// TIA Portal V16 export
// export: Created 2021-08-26T13:23:50.3138984Z, ExportSetting WithDefaults, DisplayName Totally Integrated Automation Portal, DisplayVersion V16 Update 4, DisplayName TIA Portal Version Control Interface, DisplayVersion V16 Update 2, DisplayName TIA Portal Openness, DisplayVersion V16 Update 4, DisplayName STEP 7 Professional, DisplayVersion V16 Update 4, DisplayName STEP 7 Safety, DisplayVersion V16, DisplayName WinCC Advanced, DisplayVersion V16 Update 4
FUNCTION "funkcja1" : Void   // FC1, LAD
TITLE = taki oto jest tytul bloku
{ S7_Optimized_Access := 'TRUE' }
VERSION : 0.1
// komentarz bloku
// stored: AutoNumber false, IsIECCheckEnabled false, SetENOAutomatically false, UDAEnableTagReadback false
BEGIN

REGION Network 1: bardzo ważny komentarz
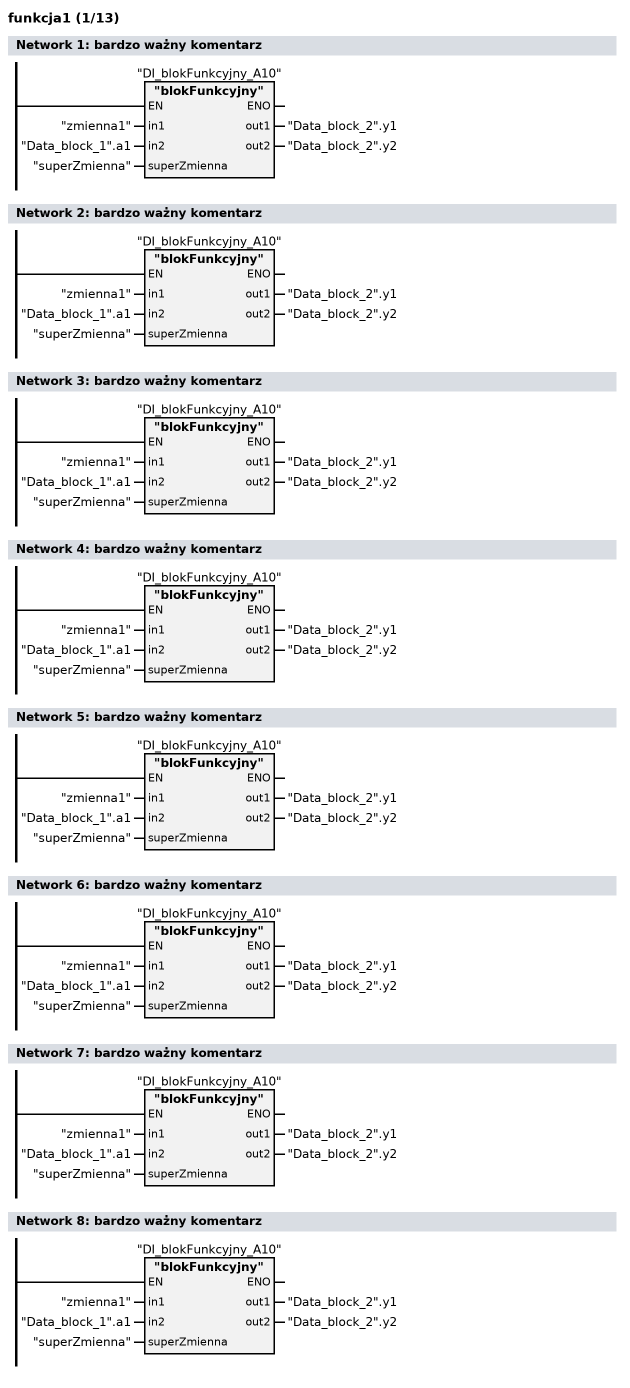
   RUNG wire#powerrail
      "DI_blokFunkcyjny_A10"(in1 := "zmienna1", in2 := "Data_block_1".a1, superZmienna := "superZmienna", out1 => "Data_block_2".y1, out2 => "Data_block_2".y2)
   END_RUNG
   // the same network as SCL:
   "DI_blokFunkcyjny_A10"(in1 := "zmienna1",   // "blokFunkcyjny"
                          in2 := "Data_block_1".a1,
                          superZmienna := "superZmienna",
                          out1 => "Data_block_2".y1,
                          out2 => "Data_block_2".y2);
END_REGION

REGION Network 2: bardzo ważny komentarz
   RUNG wire#powerrail
      "DI_blokFunkcyjny_A10"(in1 := "zmienna1", in2 := "Data_block_1".a1, superZmienna := "superZmienna", out1 => "Data_block_2".y1, out2 => "Data_block_2".y2)
   END_RUNG
   // the same network as SCL:
   "DI_blokFunkcyjny_A10"(in1 := "zmienna1",   // "blokFunkcyjny"
                          in2 := "Data_block_1".a1,
                          superZmienna := "superZmienna",
                          out1 => "Data_block_2".y1,
                          out2 => "Data_block_2".y2);
END_REGION

REGION Network 3: bardzo ważny komentarz
   RUNG wire#powerrail
      "DI_blokFunkcyjny_A10"(in1 := "zmienna1", in2 := "Data_block_1".a1, superZmienna := "superZmienna", out1 => "Data_block_2".y1, out2 => "Data_block_2".y2)
   END_RUNG
   // the same network as SCL:
   "DI_blokFunkcyjny_A10"(in1 := "zmienna1",   // "blokFunkcyjny"
                          in2 := "Data_block_1".a1,
                          superZmienna := "superZmienna",
                          out1 => "Data_block_2".y1,
                          out2 => "Data_block_2".y2);
END_REGION

REGION Network 4: bardzo ważny komentarz
   RUNG wire#powerrail
      "DI_blokFunkcyjny_A10"(in1 := "zmienna1", in2 := "Data_block_1".a1, superZmienna := "superZmienna", out1 => "Data_block_2".y1, out2 => "Data_block_2".y2)
   END_RUNG
   // the same network as SCL:
   "DI_blokFunkcyjny_A10"(in1 := "zmienna1",   // "blokFunkcyjny"
                          in2 := "Data_block_1".a1,
                          superZmienna := "superZmienna",
                          out1 => "Data_block_2".y1,
                          out2 => "Data_block_2".y2);
END_REGION

REGION Network 5: bardzo ważny komentarz
   RUNG wire#powerrail
      "DI_blokFunkcyjny_A10"(in1 := "zmienna1", in2 := "Data_block_1".a1, superZmienna := "superZmienna", out1 => "Data_block_2".y1, out2 => "Data_block_2".y2)
   END_RUNG
   // the same network as SCL:
   "DI_blokFunkcyjny_A10"(in1 := "zmienna1",   // "blokFunkcyjny"
                          in2 := "Data_block_1".a1,
                          superZmienna := "superZmienna",
                          out1 => "Data_block_2".y1,
                          out2 => "Data_block_2".y2);
END_REGION

REGION Network 6: bardzo ważny komentarz
   RUNG wire#powerrail
      "DI_blokFunkcyjny_A10"(in1 := "zmienna1", in2 := "Data_block_1".a1, superZmienna := "superZmienna", out1 => "Data_block_2".y1, out2 => "Data_block_2".y2)
   END_RUNG
   // the same network as SCL:
   "DI_blokFunkcyjny_A10"(in1 := "zmienna1",   // "blokFunkcyjny"
                          in2 := "Data_block_1".a1,
                          superZmienna := "superZmienna",
                          out1 => "Data_block_2".y1,
                          out2 => "Data_block_2".y2);
END_REGION

REGION Network 7: bardzo ważny komentarz
   RUNG wire#powerrail
      "DI_blokFunkcyjny_A10"(in1 := "zmienna1", in2 := "Data_block_1".a1, superZmienna := "superZmienna", out1 => "Data_block_2".y1, out2 => "Data_block_2".y2)
   END_RUNG
   // the same network as SCL:
   "DI_blokFunkcyjny_A10"(in1 := "zmienna1",   // "blokFunkcyjny"
                          in2 := "Data_block_1".a1,
                          superZmienna := "superZmienna",
                          out1 => "Data_block_2".y1,
                          out2 => "Data_block_2".y2);
END_REGION

REGION Network 8: bardzo ważny komentarz
   RUNG wire#powerrail
      "DI_blokFunkcyjny_A10"(in1 := "zmienna1", in2 := "Data_block_1".a1, superZmienna := "superZmienna", out1 => "Data_block_2".y1, out2 => "Data_block_2".y2)
   END_RUNG
   // the same network as SCL:
   "DI_blokFunkcyjny_A10"(in1 := "zmienna1",   // "blokFunkcyjny"
                          in2 := "Data_block_1".a1,
                          superZmienna := "superZmienna",
                          out1 => "Data_block_2".y1,
                          out2 => "Data_block_2".y2);
END_REGION

REGION Network 9: bardzo ważny komentarz
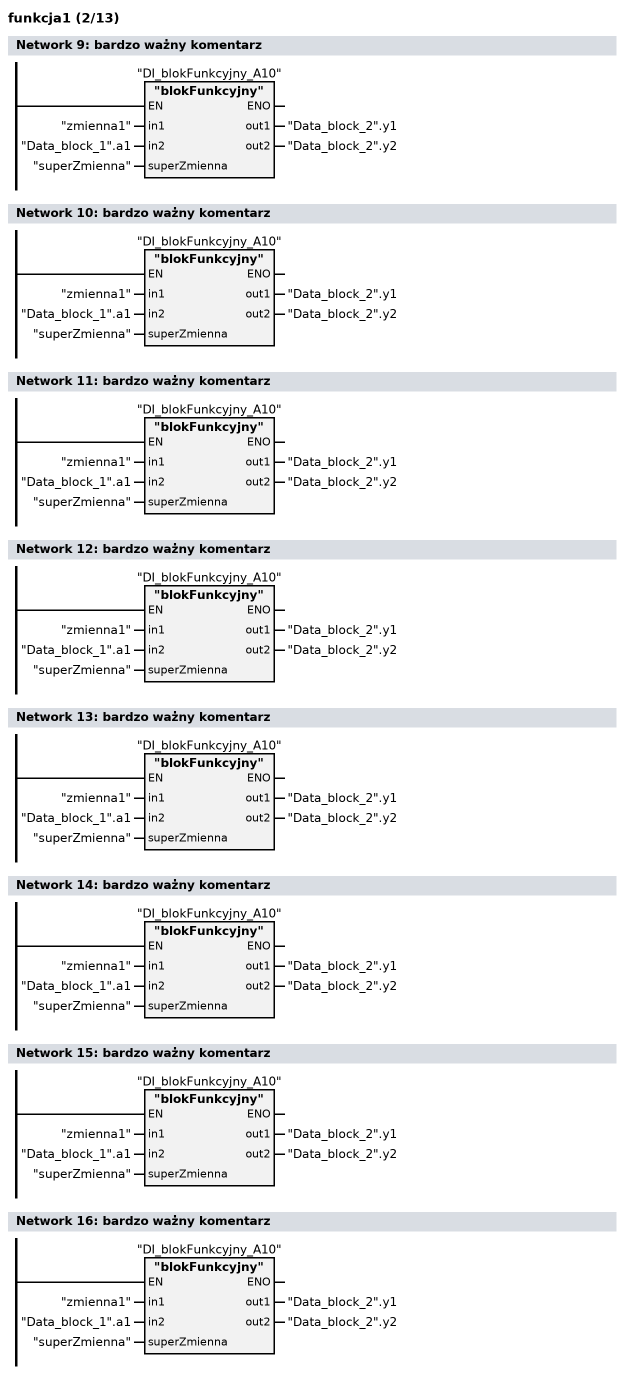
   RUNG wire#powerrail
      "DI_blokFunkcyjny_A10"(in1 := "zmienna1", in2 := "Data_block_1".a1, superZmienna := "superZmienna", out1 => "Data_block_2".y1, out2 => "Data_block_2".y2)
   END_RUNG
   // the same network as SCL:
   "DI_blokFunkcyjny_A10"(in1 := "zmienna1",   // "blokFunkcyjny"
                          in2 := "Data_block_1".a1,
                          superZmienna := "superZmienna",
                          out1 => "Data_block_2".y1,
                          out2 => "Data_block_2".y2);
END_REGION

REGION Network 10: bardzo ważny komentarz
   RUNG wire#powerrail
      "DI_blokFunkcyjny_A10"(in1 := "zmienna1", in2 := "Data_block_1".a1, superZmienna := "superZmienna", out1 => "Data_block_2".y1, out2 => "Data_block_2".y2)
   END_RUNG
   // the same network as SCL:
   "DI_blokFunkcyjny_A10"(in1 := "zmienna1",   // "blokFunkcyjny"
                          in2 := "Data_block_1".a1,
                          superZmienna := "superZmienna",
                          out1 => "Data_block_2".y1,
                          out2 => "Data_block_2".y2);
END_REGION

REGION Network 11: bardzo ważny komentarz
   RUNG wire#powerrail
      "DI_blokFunkcyjny_A10"(in1 := "zmienna1", in2 := "Data_block_1".a1, superZmienna := "superZmienna", out1 => "Data_block_2".y1, out2 => "Data_block_2".y2)
   END_RUNG
   // the same network as SCL:
   "DI_blokFunkcyjny_A10"(in1 := "zmienna1",   // "blokFunkcyjny"
                          in2 := "Data_block_1".a1,
                          superZmienna := "superZmienna",
                          out1 => "Data_block_2".y1,
                          out2 => "Data_block_2".y2);
END_REGION

REGION Network 12: bardzo ważny komentarz
   RUNG wire#powerrail
      "DI_blokFunkcyjny_A10"(in1 := "zmienna1", in2 := "Data_block_1".a1, superZmienna := "superZmienna", out1 => "Data_block_2".y1, out2 => "Data_block_2".y2)
   END_RUNG
   // the same network as SCL:
   "DI_blokFunkcyjny_A10"(in1 := "zmienna1",   // "blokFunkcyjny"
                          in2 := "Data_block_1".a1,
                          superZmienna := "superZmienna",
                          out1 => "Data_block_2".y1,
                          out2 => "Data_block_2".y2);
END_REGION

REGION Network 13: bardzo ważny komentarz
   RUNG wire#powerrail
      "DI_blokFunkcyjny_A10"(in1 := "zmienna1", in2 := "Data_block_1".a1, superZmienna := "superZmienna", out1 => "Data_block_2".y1, out2 => "Data_block_2".y2)
   END_RUNG
   // the same network as SCL:
   "DI_blokFunkcyjny_A10"(in1 := "zmienna1",   // "blokFunkcyjny"
                          in2 := "Data_block_1".a1,
                          superZmienna := "superZmienna",
                          out1 => "Data_block_2".y1,
                          out2 => "Data_block_2".y2);
END_REGION

REGION Network 14: bardzo ważny komentarz
   RUNG wire#powerrail
      "DI_blokFunkcyjny_A10"(in1 := "zmienna1", in2 := "Data_block_1".a1, superZmienna := "superZmienna", out1 => "Data_block_2".y1, out2 => "Data_block_2".y2)
   END_RUNG
   // the same network as SCL:
   "DI_blokFunkcyjny_A10"(in1 := "zmienna1",   // "blokFunkcyjny"
                          in2 := "Data_block_1".a1,
                          superZmienna := "superZmienna",
                          out1 => "Data_block_2".y1,
                          out2 => "Data_block_2".y2);
END_REGION

REGION Network 15: bardzo ważny komentarz
   RUNG wire#powerrail
      "DI_blokFunkcyjny_A10"(in1 := "zmienna1", in2 := "Data_block_1".a1, superZmienna := "superZmienna", out1 => "Data_block_2".y1, out2 => "Data_block_2".y2)
   END_RUNG
   // the same network as SCL:
   "DI_blokFunkcyjny_A10"(in1 := "zmienna1",   // "blokFunkcyjny"
                          in2 := "Data_block_1".a1,
                          superZmienna := "superZmienna",
                          out1 => "Data_block_2".y1,
                          out2 => "Data_block_2".y2);
END_REGION

REGION Network 16: bardzo ważny komentarz
   RUNG wire#powerrail
      "DI_blokFunkcyjny_A10"(in1 := "zmienna1", in2 := "Data_block_1".a1, superZmienna := "superZmienna", out1 => "Data_block_2".y1, out2 => "Data_block_2".y2)
   END_RUNG
   // the same network as SCL:
   "DI_blokFunkcyjny_A10"(in1 := "zmienna1",   // "blokFunkcyjny"
                          in2 := "Data_block_1".a1,
                          superZmienna := "superZmienna",
                          out1 => "Data_block_2".y1,
                          out2 => "Data_block_2".y2);
END_REGION

REGION Network 17: bardzo ważny komentarz
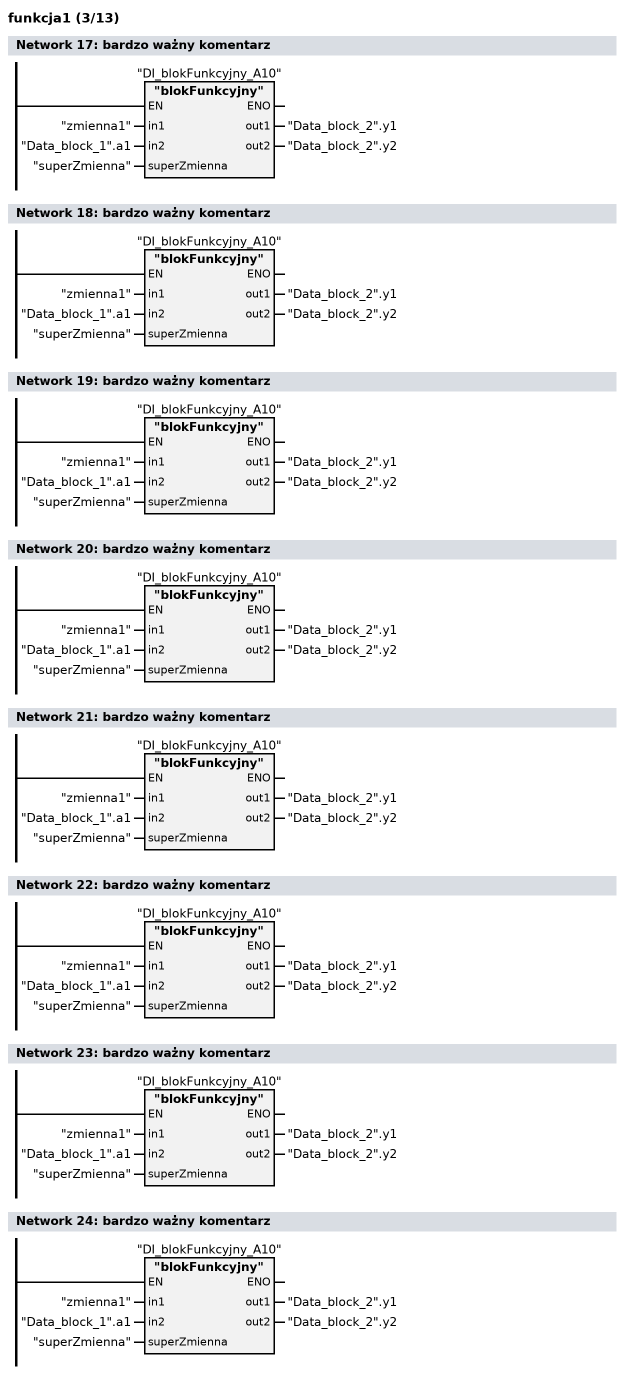
   RUNG wire#powerrail
      "DI_blokFunkcyjny_A10"(in1 := "zmienna1", in2 := "Data_block_1".a1, superZmienna := "superZmienna", out1 => "Data_block_2".y1, out2 => "Data_block_2".y2)
   END_RUNG
   // the same network as SCL:
   "DI_blokFunkcyjny_A10"(in1 := "zmienna1",   // "blokFunkcyjny"
                          in2 := "Data_block_1".a1,
                          superZmienna := "superZmienna",
                          out1 => "Data_block_2".y1,
                          out2 => "Data_block_2".y2);
END_REGION

REGION Network 18: bardzo ważny komentarz
   RUNG wire#powerrail
      "DI_blokFunkcyjny_A10"(in1 := "zmienna1", in2 := "Data_block_1".a1, superZmienna := "superZmienna", out1 => "Data_block_2".y1, out2 => "Data_block_2".y2)
   END_RUNG
   // the same network as SCL:
   "DI_blokFunkcyjny_A10"(in1 := "zmienna1",   // "blokFunkcyjny"
                          in2 := "Data_block_1".a1,
                          superZmienna := "superZmienna",
                          out1 => "Data_block_2".y1,
                          out2 => "Data_block_2".y2);
END_REGION

REGION Network 19: bardzo ważny komentarz
   RUNG wire#powerrail
      "DI_blokFunkcyjny_A10"(in1 := "zmienna1", in2 := "Data_block_1".a1, superZmienna := "superZmienna", out1 => "Data_block_2".y1, out2 => "Data_block_2".y2)
   END_RUNG
   // the same network as SCL:
   "DI_blokFunkcyjny_A10"(in1 := "zmienna1",   // "blokFunkcyjny"
                          in2 := "Data_block_1".a1,
                          superZmienna := "superZmienna",
                          out1 => "Data_block_2".y1,
                          out2 => "Data_block_2".y2);
END_REGION

REGION Network 20: bardzo ważny komentarz
   RUNG wire#powerrail
      "DI_blokFunkcyjny_A10"(in1 := "zmienna1", in2 := "Data_block_1".a1, superZmienna := "superZmienna", out1 => "Data_block_2".y1, out2 => "Data_block_2".y2)
   END_RUNG
   // the same network as SCL:
   "DI_blokFunkcyjny_A10"(in1 := "zmienna1",   // "blokFunkcyjny"
                          in2 := "Data_block_1".a1,
                          superZmienna := "superZmienna",
                          out1 => "Data_block_2".y1,
                          out2 => "Data_block_2".y2);
END_REGION

REGION Network 21: bardzo ważny komentarz
   RUNG wire#powerrail
      "DI_blokFunkcyjny_A10"(in1 := "zmienna1", in2 := "Data_block_1".a1, superZmienna := "superZmienna", out1 => "Data_block_2".y1, out2 => "Data_block_2".y2)
   END_RUNG
   // the same network as SCL:
   "DI_blokFunkcyjny_A10"(in1 := "zmienna1",   // "blokFunkcyjny"
                          in2 := "Data_block_1".a1,
                          superZmienna := "superZmienna",
                          out1 => "Data_block_2".y1,
                          out2 => "Data_block_2".y2);
END_REGION

REGION Network 22: bardzo ważny komentarz
   RUNG wire#powerrail
      "DI_blokFunkcyjny_A10"(in1 := "zmienna1", in2 := "Data_block_1".a1, superZmienna := "superZmienna", out1 => "Data_block_2".y1, out2 => "Data_block_2".y2)
   END_RUNG
   // the same network as SCL:
   "DI_blokFunkcyjny_A10"(in1 := "zmienna1",   // "blokFunkcyjny"
                          in2 := "Data_block_1".a1,
                          superZmienna := "superZmienna",
                          out1 => "Data_block_2".y1,
                          out2 => "Data_block_2".y2);
END_REGION

REGION Network 23: bardzo ważny komentarz
   RUNG wire#powerrail
      "DI_blokFunkcyjny_A10"(in1 := "zmienna1", in2 := "Data_block_1".a1, superZmienna := "superZmienna", out1 => "Data_block_2".y1, out2 => "Data_block_2".y2)
   END_RUNG
   // the same network as SCL:
   "DI_blokFunkcyjny_A10"(in1 := "zmienna1",   // "blokFunkcyjny"
                          in2 := "Data_block_1".a1,
                          superZmienna := "superZmienna",
                          out1 => "Data_block_2".y1,
                          out2 => "Data_block_2".y2);
END_REGION

REGION Network 24: bardzo ważny komentarz
   RUNG wire#powerrail
      "DI_blokFunkcyjny_A10"(in1 := "zmienna1", in2 := "Data_block_1".a1, superZmienna := "superZmienna", out1 => "Data_block_2".y1, out2 => "Data_block_2".y2)
   END_RUNG
   // the same network as SCL:
   "DI_blokFunkcyjny_A10"(in1 := "zmienna1",   // "blokFunkcyjny"
                          in2 := "Data_block_1".a1,
                          superZmienna := "superZmienna",
                          out1 => "Data_block_2".y1,
                          out2 => "Data_block_2".y2);
END_REGION

REGION Network 25: bardzo ważny komentarz
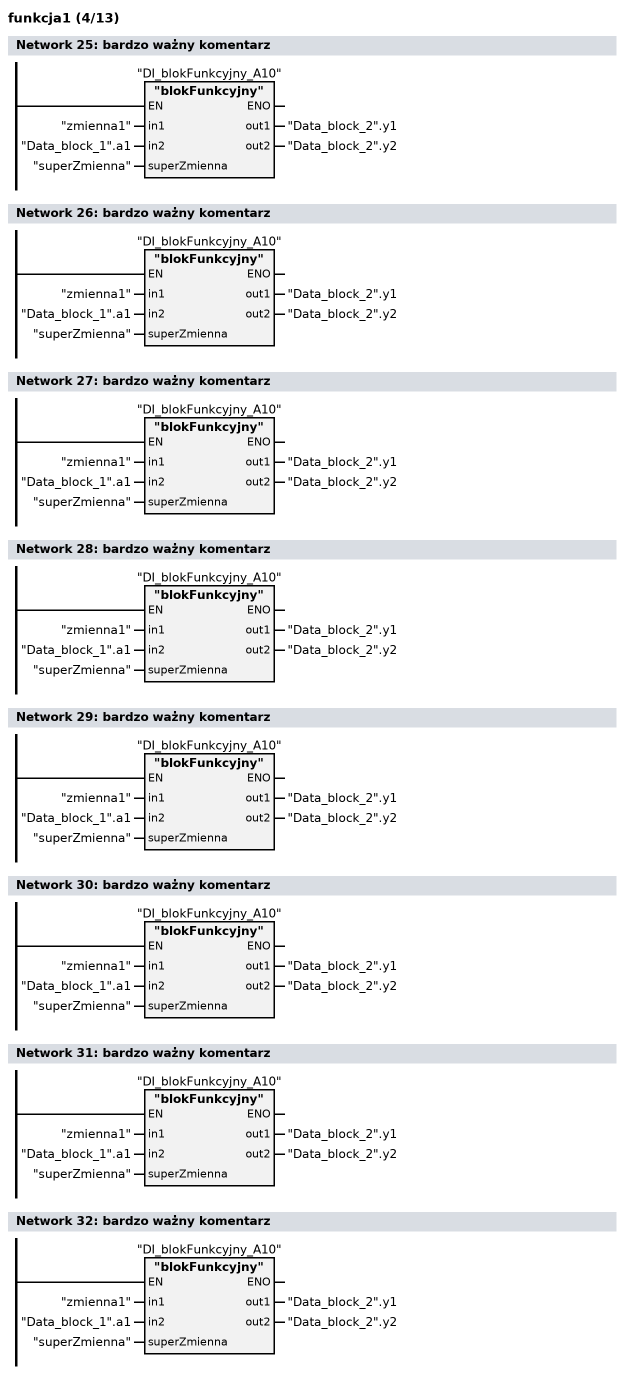
   RUNG wire#powerrail
      "DI_blokFunkcyjny_A10"(in1 := "zmienna1", in2 := "Data_block_1".a1, superZmienna := "superZmienna", out1 => "Data_block_2".y1, out2 => "Data_block_2".y2)
   END_RUNG
   // the same network as SCL:
   "DI_blokFunkcyjny_A10"(in1 := "zmienna1",   // "blokFunkcyjny"
                          in2 := "Data_block_1".a1,
                          superZmienna := "superZmienna",
                          out1 => "Data_block_2".y1,
                          out2 => "Data_block_2".y2);
END_REGION

REGION Network 26: bardzo ważny komentarz
   RUNG wire#powerrail
      "DI_blokFunkcyjny_A10"(in1 := "zmienna1", in2 := "Data_block_1".a1, superZmienna := "superZmienna", out1 => "Data_block_2".y1, out2 => "Data_block_2".y2)
   END_RUNG
   // the same network as SCL:
   "DI_blokFunkcyjny_A10"(in1 := "zmienna1",   // "blokFunkcyjny"
                          in2 := "Data_block_1".a1,
                          superZmienna := "superZmienna",
                          out1 => "Data_block_2".y1,
                          out2 => "Data_block_2".y2);
END_REGION

REGION Network 27: bardzo ważny komentarz
   RUNG wire#powerrail
      "DI_blokFunkcyjny_A10"(in1 := "zmienna1", in2 := "Data_block_1".a1, superZmienna := "superZmienna", out1 => "Data_block_2".y1, out2 => "Data_block_2".y2)
   END_RUNG
   // the same network as SCL:
   "DI_blokFunkcyjny_A10"(in1 := "zmienna1",   // "blokFunkcyjny"
                          in2 := "Data_block_1".a1,
                          superZmienna := "superZmienna",
                          out1 => "Data_block_2".y1,
                          out2 => "Data_block_2".y2);
END_REGION

REGION Network 28: bardzo ważny komentarz
   RUNG wire#powerrail
      "DI_blokFunkcyjny_A10"(in1 := "zmienna1", in2 := "Data_block_1".a1, superZmienna := "superZmienna", out1 => "Data_block_2".y1, out2 => "Data_block_2".y2)
   END_RUNG
   // the same network as SCL:
   "DI_blokFunkcyjny_A10"(in1 := "zmienna1",   // "blokFunkcyjny"
                          in2 := "Data_block_1".a1,
                          superZmienna := "superZmienna",
                          out1 => "Data_block_2".y1,
                          out2 => "Data_block_2".y2);
END_REGION

REGION Network 29: bardzo ważny komentarz
   RUNG wire#powerrail
      "DI_blokFunkcyjny_A10"(in1 := "zmienna1", in2 := "Data_block_1".a1, superZmienna := "superZmienna", out1 => "Data_block_2".y1, out2 => "Data_block_2".y2)
   END_RUNG
   // the same network as SCL:
   "DI_blokFunkcyjny_A10"(in1 := "zmienna1",   // "blokFunkcyjny"
                          in2 := "Data_block_1".a1,
                          superZmienna := "superZmienna",
                          out1 => "Data_block_2".y1,
                          out2 => "Data_block_2".y2);
END_REGION

REGION Network 30: bardzo ważny komentarz
   RUNG wire#powerrail
      "DI_blokFunkcyjny_A10"(in1 := "zmienna1", in2 := "Data_block_1".a1, superZmienna := "superZmienna", out1 => "Data_block_2".y1, out2 => "Data_block_2".y2)
   END_RUNG
   // the same network as SCL:
   "DI_blokFunkcyjny_A10"(in1 := "zmienna1",   // "blokFunkcyjny"
                          in2 := "Data_block_1".a1,
                          superZmienna := "superZmienna",
                          out1 => "Data_block_2".y1,
                          out2 => "Data_block_2".y2);
END_REGION

REGION Network 31: bardzo ważny komentarz
   RUNG wire#powerrail
      "DI_blokFunkcyjny_A10"(in1 := "zmienna1", in2 := "Data_block_1".a1, superZmienna := "superZmienna", out1 => "Data_block_2".y1, out2 => "Data_block_2".y2)
   END_RUNG
   // the same network as SCL:
   "DI_blokFunkcyjny_A10"(in1 := "zmienna1",   // "blokFunkcyjny"
                          in2 := "Data_block_1".a1,
                          superZmienna := "superZmienna",
                          out1 => "Data_block_2".y1,
                          out2 => "Data_block_2".y2);
END_REGION

REGION Network 32: bardzo ważny komentarz
   RUNG wire#powerrail
      "DI_blokFunkcyjny_A10"(in1 := "zmienna1", in2 := "Data_block_1".a1, superZmienna := "superZmienna", out1 => "Data_block_2".y1, out2 => "Data_block_2".y2)
   END_RUNG
   // the same network as SCL:
   "DI_blokFunkcyjny_A10"(in1 := "zmienna1",   // "blokFunkcyjny"
                          in2 := "Data_block_1".a1,
                          superZmienna := "superZmienna",
                          out1 => "Data_block_2".y1,
                          out2 => "Data_block_2".y2);
END_REGION

REGION Network 33: bardzo ważny komentarz
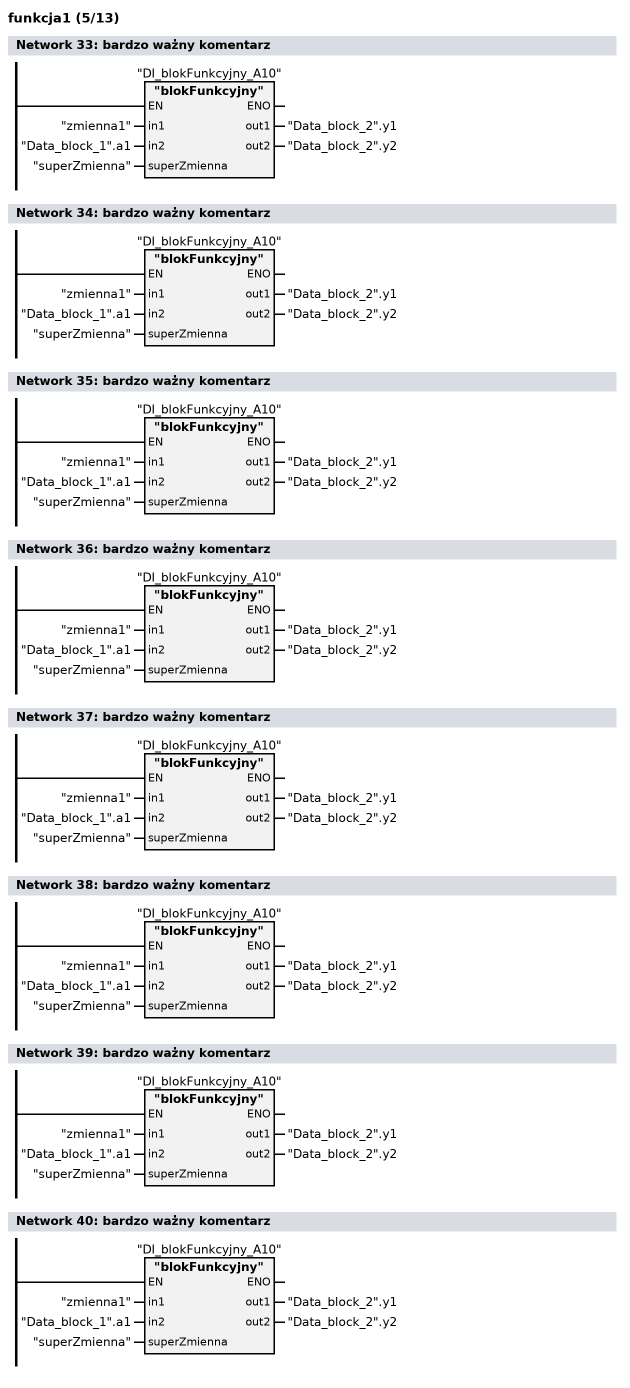
   RUNG wire#powerrail
      "DI_blokFunkcyjny_A10"(in1 := "zmienna1", in2 := "Data_block_1".a1, superZmienna := "superZmienna", out1 => "Data_block_2".y1, out2 => "Data_block_2".y2)
   END_RUNG
   // the same network as SCL:
   "DI_blokFunkcyjny_A10"(in1 := "zmienna1",   // "blokFunkcyjny"
                          in2 := "Data_block_1".a1,
                          superZmienna := "superZmienna",
                          out1 => "Data_block_2".y1,
                          out2 => "Data_block_2".y2);
END_REGION

REGION Network 34: bardzo ważny komentarz
   RUNG wire#powerrail
      "DI_blokFunkcyjny_A10"(in1 := "zmienna1", in2 := "Data_block_1".a1, superZmienna := "superZmienna", out1 => "Data_block_2".y1, out2 => "Data_block_2".y2)
   END_RUNG
   // the same network as SCL:
   "DI_blokFunkcyjny_A10"(in1 := "zmienna1",   // "blokFunkcyjny"
                          in2 := "Data_block_1".a1,
                          superZmienna := "superZmienna",
                          out1 => "Data_block_2".y1,
                          out2 => "Data_block_2".y2);
END_REGION

REGION Network 35: bardzo ważny komentarz
   RUNG wire#powerrail
      "DI_blokFunkcyjny_A10"(in1 := "zmienna1", in2 := "Data_block_1".a1, superZmienna := "superZmienna", out1 => "Data_block_2".y1, out2 => "Data_block_2".y2)
   END_RUNG
   // the same network as SCL:
   "DI_blokFunkcyjny_A10"(in1 := "zmienna1",   // "blokFunkcyjny"
                          in2 := "Data_block_1".a1,
                          superZmienna := "superZmienna",
                          out1 => "Data_block_2".y1,
                          out2 => "Data_block_2".y2);
END_REGION

REGION Network 36: bardzo ważny komentarz
   RUNG wire#powerrail
      "DI_blokFunkcyjny_A10"(in1 := "zmienna1", in2 := "Data_block_1".a1, superZmienna := "superZmienna", out1 => "Data_block_2".y1, out2 => "Data_block_2".y2)
   END_RUNG
   // the same network as SCL:
   "DI_blokFunkcyjny_A10"(in1 := "zmienna1",   // "blokFunkcyjny"
                          in2 := "Data_block_1".a1,
                          superZmienna := "superZmienna",
                          out1 => "Data_block_2".y1,
                          out2 => "Data_block_2".y2);
END_REGION

REGION Network 37: bardzo ważny komentarz
   RUNG wire#powerrail
      "DI_blokFunkcyjny_A10"(in1 := "zmienna1", in2 := "Data_block_1".a1, superZmienna := "superZmienna", out1 => "Data_block_2".y1, out2 => "Data_block_2".y2)
   END_RUNG
   // the same network as SCL:
   "DI_blokFunkcyjny_A10"(in1 := "zmienna1",   // "blokFunkcyjny"
                          in2 := "Data_block_1".a1,
                          superZmienna := "superZmienna",
                          out1 => "Data_block_2".y1,
                          out2 => "Data_block_2".y2);
END_REGION

REGION Network 38: bardzo ważny komentarz
   RUNG wire#powerrail
      "DI_blokFunkcyjny_A10"(in1 := "zmienna1", in2 := "Data_block_1".a1, superZmienna := "superZmienna", out1 => "Data_block_2".y1, out2 => "Data_block_2".y2)
   END_RUNG
   // the same network as SCL:
   "DI_blokFunkcyjny_A10"(in1 := "zmienna1",   // "blokFunkcyjny"
                          in2 := "Data_block_1".a1,
                          superZmienna := "superZmienna",
                          out1 => "Data_block_2".y1,
                          out2 => "Data_block_2".y2);
END_REGION

REGION Network 39: bardzo ważny komentarz
   RUNG wire#powerrail
      "DI_blokFunkcyjny_A10"(in1 := "zmienna1", in2 := "Data_block_1".a1, superZmienna := "superZmienna", out1 => "Data_block_2".y1, out2 => "Data_block_2".y2)
   END_RUNG
   // the same network as SCL:
   "DI_blokFunkcyjny_A10"(in1 := "zmienna1",   // "blokFunkcyjny"
                          in2 := "Data_block_1".a1,
                          superZmienna := "superZmienna",
                          out1 => "Data_block_2".y1,
                          out2 => "Data_block_2".y2);
END_REGION

REGION Network 40: bardzo ważny komentarz
   RUNG wire#powerrail
      "DI_blokFunkcyjny_A10"(in1 := "zmienna1", in2 := "Data_block_1".a1, superZmienna := "superZmienna", out1 => "Data_block_2".y1, out2 => "Data_block_2".y2)
   END_RUNG
   // the same network as SCL:
   "DI_blokFunkcyjny_A10"(in1 := "zmienna1",   // "blokFunkcyjny"
                          in2 := "Data_block_1".a1,
                          superZmienna := "superZmienna",
                          out1 => "Data_block_2".y1,
                          out2 => "Data_block_2".y2);
END_REGION

REGION Network 41: bardzo ważny komentarz
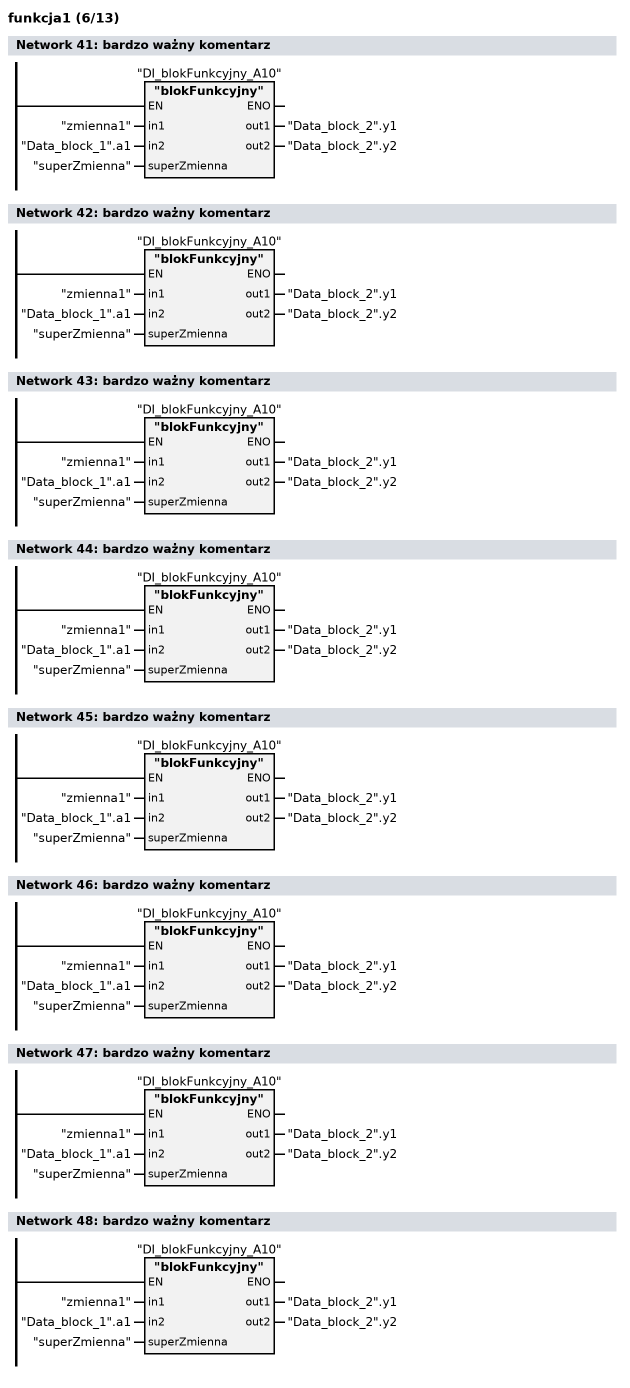
   RUNG wire#powerrail
      "DI_blokFunkcyjny_A10"(in1 := "zmienna1", in2 := "Data_block_1".a1, superZmienna := "superZmienna", out1 => "Data_block_2".y1, out2 => "Data_block_2".y2)
   END_RUNG
   // the same network as SCL:
   "DI_blokFunkcyjny_A10"(in1 := "zmienna1",   // "blokFunkcyjny"
                          in2 := "Data_block_1".a1,
                          superZmienna := "superZmienna",
                          out1 => "Data_block_2".y1,
                          out2 => "Data_block_2".y2);
END_REGION

REGION Network 42: bardzo ważny komentarz
   RUNG wire#powerrail
      "DI_blokFunkcyjny_A10"(in1 := "zmienna1", in2 := "Data_block_1".a1, superZmienna := "superZmienna", out1 => "Data_block_2".y1, out2 => "Data_block_2".y2)
   END_RUNG
   // the same network as SCL:
   "DI_blokFunkcyjny_A10"(in1 := "zmienna1",   // "blokFunkcyjny"
                          in2 := "Data_block_1".a1,
                          superZmienna := "superZmienna",
                          out1 => "Data_block_2".y1,
                          out2 => "Data_block_2".y2);
END_REGION

REGION Network 43: bardzo ważny komentarz
   RUNG wire#powerrail
      "DI_blokFunkcyjny_A10"(in1 := "zmienna1", in2 := "Data_block_1".a1, superZmienna := "superZmienna", out1 => "Data_block_2".y1, out2 => "Data_block_2".y2)
   END_RUNG
   // the same network as SCL:
   "DI_blokFunkcyjny_A10"(in1 := "zmienna1",   // "blokFunkcyjny"
                          in2 := "Data_block_1".a1,
                          superZmienna := "superZmienna",
                          out1 => "Data_block_2".y1,
                          out2 => "Data_block_2".y2);
END_REGION

REGION Network 44: bardzo ważny komentarz
   RUNG wire#powerrail
      "DI_blokFunkcyjny_A10"(in1 := "zmienna1", in2 := "Data_block_1".a1, superZmienna := "superZmienna", out1 => "Data_block_2".y1, out2 => "Data_block_2".y2)
   END_RUNG
   // the same network as SCL:
   "DI_blokFunkcyjny_A10"(in1 := "zmienna1",   // "blokFunkcyjny"
                          in2 := "Data_block_1".a1,
                          superZmienna := "superZmienna",
                          out1 => "Data_block_2".y1,
                          out2 => "Data_block_2".y2);
END_REGION

REGION Network 45: bardzo ważny komentarz
   RUNG wire#powerrail
      "DI_blokFunkcyjny_A10"(in1 := "zmienna1", in2 := "Data_block_1".a1, superZmienna := "superZmienna", out1 => "Data_block_2".y1, out2 => "Data_block_2".y2)
   END_RUNG
   // the same network as SCL:
   "DI_blokFunkcyjny_A10"(in1 := "zmienna1",   // "blokFunkcyjny"
                          in2 := "Data_block_1".a1,
                          superZmienna := "superZmienna",
                          out1 => "Data_block_2".y1,
                          out2 => "Data_block_2".y2);
END_REGION

REGION Network 46: bardzo ważny komentarz
   RUNG wire#powerrail
      "DI_blokFunkcyjny_A10"(in1 := "zmienna1", in2 := "Data_block_1".a1, superZmienna := "superZmienna", out1 => "Data_block_2".y1, out2 => "Data_block_2".y2)
   END_RUNG
   // the same network as SCL:
   "DI_blokFunkcyjny_A10"(in1 := "zmienna1",   // "blokFunkcyjny"
                          in2 := "Data_block_1".a1,
                          superZmienna := "superZmienna",
                          out1 => "Data_block_2".y1,
                          out2 => "Data_block_2".y2);
END_REGION

REGION Network 47: bardzo ważny komentarz
   RUNG wire#powerrail
      "DI_blokFunkcyjny_A10"(in1 := "zmienna1", in2 := "Data_block_1".a1, superZmienna := "superZmienna", out1 => "Data_block_2".y1, out2 => "Data_block_2".y2)
   END_RUNG
   // the same network as SCL:
   "DI_blokFunkcyjny_A10"(in1 := "zmienna1",   // "blokFunkcyjny"
                          in2 := "Data_block_1".a1,
                          superZmienna := "superZmienna",
                          out1 => "Data_block_2".y1,
                          out2 => "Data_block_2".y2);
END_REGION

REGION Network 48: bardzo ważny komentarz
   RUNG wire#powerrail
      "DI_blokFunkcyjny_A10"(in1 := "zmienna1", in2 := "Data_block_1".a1, superZmienna := "superZmienna", out1 => "Data_block_2".y1, out2 => "Data_block_2".y2)
   END_RUNG
   // the same network as SCL:
   "DI_blokFunkcyjny_A10"(in1 := "zmienna1",   // "blokFunkcyjny"
                          in2 := "Data_block_1".a1,
                          superZmienna := "superZmienna",
                          out1 => "Data_block_2".y1,
                          out2 => "Data_block_2".y2);
END_REGION

REGION Network 49: bardzo ważny komentarz
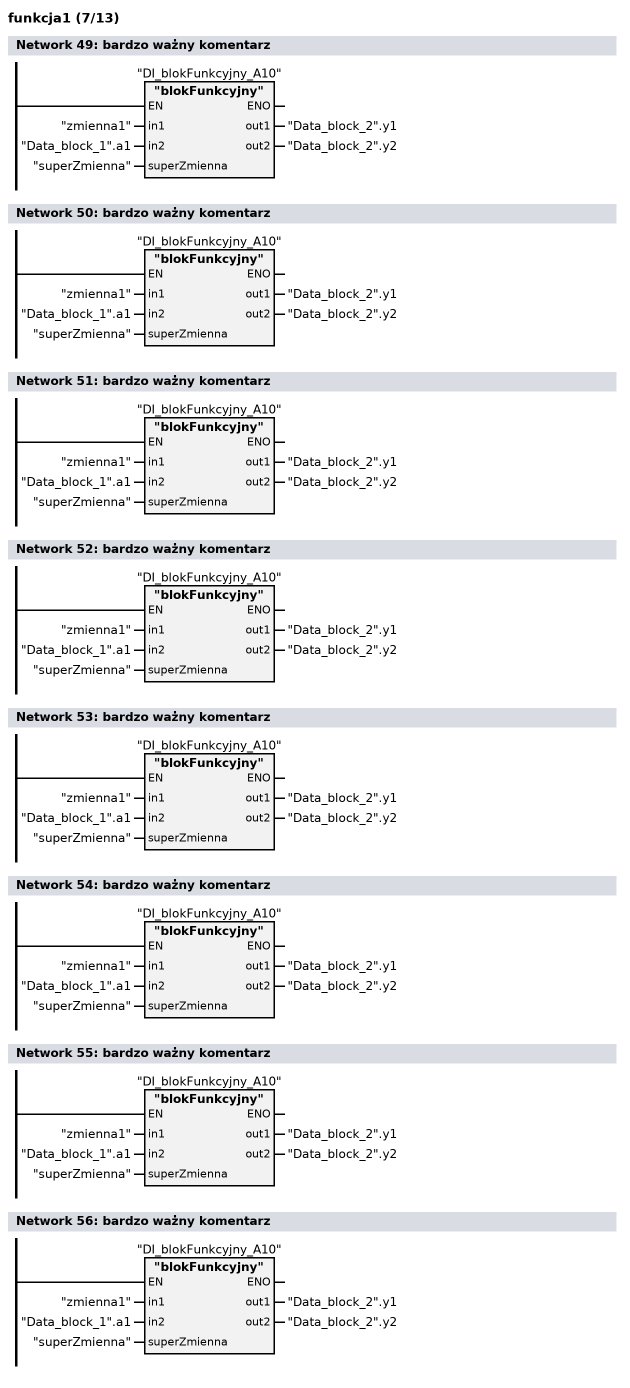
   RUNG wire#powerrail
      "DI_blokFunkcyjny_A10"(in1 := "zmienna1", in2 := "Data_block_1".a1, superZmienna := "superZmienna", out1 => "Data_block_2".y1, out2 => "Data_block_2".y2)
   END_RUNG
   // the same network as SCL:
   "DI_blokFunkcyjny_A10"(in1 := "zmienna1",   // "blokFunkcyjny"
                          in2 := "Data_block_1".a1,
                          superZmienna := "superZmienna",
                          out1 => "Data_block_2".y1,
                          out2 => "Data_block_2".y2);
END_REGION

REGION Network 50: bardzo ważny komentarz
   RUNG wire#powerrail
      "DI_blokFunkcyjny_A10"(in1 := "zmienna1", in2 := "Data_block_1".a1, superZmienna := "superZmienna", out1 => "Data_block_2".y1, out2 => "Data_block_2".y2)
   END_RUNG
   // the same network as SCL:
   "DI_blokFunkcyjny_A10"(in1 := "zmienna1",   // "blokFunkcyjny"
                          in2 := "Data_block_1".a1,
                          superZmienna := "superZmienna",
                          out1 => "Data_block_2".y1,
                          out2 => "Data_block_2".y2);
END_REGION

REGION Network 51: bardzo ważny komentarz
   RUNG wire#powerrail
      "DI_blokFunkcyjny_A10"(in1 := "zmienna1", in2 := "Data_block_1".a1, superZmienna := "superZmienna", out1 => "Data_block_2".y1, out2 => "Data_block_2".y2)
   END_RUNG
   // the same network as SCL:
   "DI_blokFunkcyjny_A10"(in1 := "zmienna1",   // "blokFunkcyjny"
                          in2 := "Data_block_1".a1,
                          superZmienna := "superZmienna",
                          out1 => "Data_block_2".y1,
                          out2 => "Data_block_2".y2);
END_REGION

REGION Network 52: bardzo ważny komentarz
   RUNG wire#powerrail
      "DI_blokFunkcyjny_A10"(in1 := "zmienna1", in2 := "Data_block_1".a1, superZmienna := "superZmienna", out1 => "Data_block_2".y1, out2 => "Data_block_2".y2)
   END_RUNG
   // the same network as SCL:
   "DI_blokFunkcyjny_A10"(in1 := "zmienna1",   // "blokFunkcyjny"
                          in2 := "Data_block_1".a1,
                          superZmienna := "superZmienna",
                          out1 => "Data_block_2".y1,
                          out2 => "Data_block_2".y2);
END_REGION

REGION Network 53: bardzo ważny komentarz
   RUNG wire#powerrail
      "DI_blokFunkcyjny_A10"(in1 := "zmienna1", in2 := "Data_block_1".a1, superZmienna := "superZmienna", out1 => "Data_block_2".y1, out2 => "Data_block_2".y2)
   END_RUNG
   // the same network as SCL:
   "DI_blokFunkcyjny_A10"(in1 := "zmienna1",   // "blokFunkcyjny"
                          in2 := "Data_block_1".a1,
                          superZmienna := "superZmienna",
                          out1 => "Data_block_2".y1,
                          out2 => "Data_block_2".y2);
END_REGION

REGION Network 54: bardzo ważny komentarz
   RUNG wire#powerrail
      "DI_blokFunkcyjny_A10"(in1 := "zmienna1", in2 := "Data_block_1".a1, superZmienna := "superZmienna", out1 => "Data_block_2".y1, out2 => "Data_block_2".y2)
   END_RUNG
   // the same network as SCL:
   "DI_blokFunkcyjny_A10"(in1 := "zmienna1",   // "blokFunkcyjny"
                          in2 := "Data_block_1".a1,
                          superZmienna := "superZmienna",
                          out1 => "Data_block_2".y1,
                          out2 => "Data_block_2".y2);
END_REGION

REGION Network 55: bardzo ważny komentarz
   RUNG wire#powerrail
      "DI_blokFunkcyjny_A10"(in1 := "zmienna1", in2 := "Data_block_1".a1, superZmienna := "superZmienna", out1 => "Data_block_2".y1, out2 => "Data_block_2".y2)
   END_RUNG
   // the same network as SCL:
   "DI_blokFunkcyjny_A10"(in1 := "zmienna1",   // "blokFunkcyjny"
                          in2 := "Data_block_1".a1,
                          superZmienna := "superZmienna",
                          out1 => "Data_block_2".y1,
                          out2 => "Data_block_2".y2);
END_REGION

REGION Network 56: bardzo ważny komentarz
   RUNG wire#powerrail
      "DI_blokFunkcyjny_A10"(in1 := "zmienna1", in2 := "Data_block_1".a1, superZmienna := "superZmienna", out1 => "Data_block_2".y1, out2 => "Data_block_2".y2)
   END_RUNG
   // the same network as SCL:
   "DI_blokFunkcyjny_A10"(in1 := "zmienna1",   // "blokFunkcyjny"
                          in2 := "Data_block_1".a1,
                          superZmienna := "superZmienna",
                          out1 => "Data_block_2".y1,
                          out2 => "Data_block_2".y2);
END_REGION

REGION Network 57: bardzo ważny komentarz
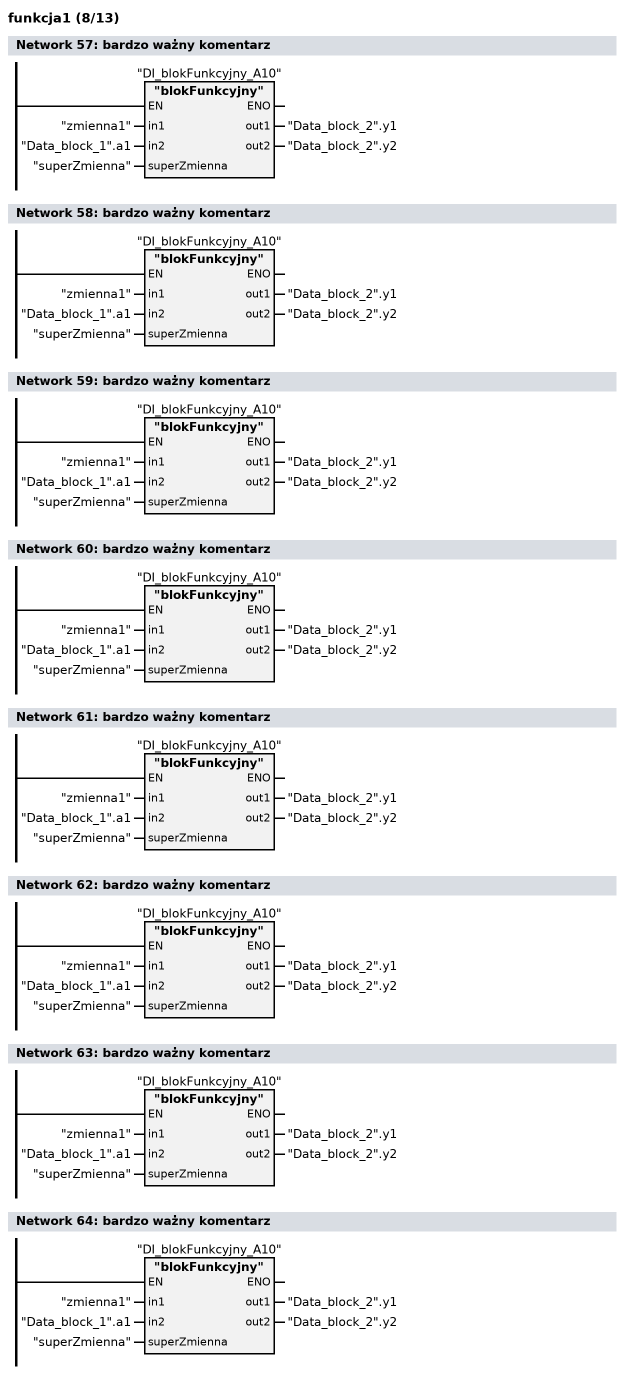
   RUNG wire#powerrail
      "DI_blokFunkcyjny_A10"(in1 := "zmienna1", in2 := "Data_block_1".a1, superZmienna := "superZmienna", out1 => "Data_block_2".y1, out2 => "Data_block_2".y2)
   END_RUNG
   // the same network as SCL:
   "DI_blokFunkcyjny_A10"(in1 := "zmienna1",   // "blokFunkcyjny"
                          in2 := "Data_block_1".a1,
                          superZmienna := "superZmienna",
                          out1 => "Data_block_2".y1,
                          out2 => "Data_block_2".y2);
END_REGION

REGION Network 58: bardzo ważny komentarz
   RUNG wire#powerrail
      "DI_blokFunkcyjny_A10"(in1 := "zmienna1", in2 := "Data_block_1".a1, superZmienna := "superZmienna", out1 => "Data_block_2".y1, out2 => "Data_block_2".y2)
   END_RUNG
   // the same network as SCL:
   "DI_blokFunkcyjny_A10"(in1 := "zmienna1",   // "blokFunkcyjny"
                          in2 := "Data_block_1".a1,
                          superZmienna := "superZmienna",
                          out1 => "Data_block_2".y1,
                          out2 => "Data_block_2".y2);
END_REGION

REGION Network 59: bardzo ważny komentarz
   RUNG wire#powerrail
      "DI_blokFunkcyjny_A10"(in1 := "zmienna1", in2 := "Data_block_1".a1, superZmienna := "superZmienna", out1 => "Data_block_2".y1, out2 => "Data_block_2".y2)
   END_RUNG
   // the same network as SCL:
   "DI_blokFunkcyjny_A10"(in1 := "zmienna1",   // "blokFunkcyjny"
                          in2 := "Data_block_1".a1,
                          superZmienna := "superZmienna",
                          out1 => "Data_block_2".y1,
                          out2 => "Data_block_2".y2);
END_REGION

REGION Network 60: bardzo ważny komentarz
   RUNG wire#powerrail
      "DI_blokFunkcyjny_A10"(in1 := "zmienna1", in2 := "Data_block_1".a1, superZmienna := "superZmienna", out1 => "Data_block_2".y1, out2 => "Data_block_2".y2)
   END_RUNG
   // the same network as SCL:
   "DI_blokFunkcyjny_A10"(in1 := "zmienna1",   // "blokFunkcyjny"
                          in2 := "Data_block_1".a1,
                          superZmienna := "superZmienna",
                          out1 => "Data_block_2".y1,
                          out2 => "Data_block_2".y2);
END_REGION

REGION Network 61: bardzo ważny komentarz
   RUNG wire#powerrail
      "DI_blokFunkcyjny_A10"(in1 := "zmienna1", in2 := "Data_block_1".a1, superZmienna := "superZmienna", out1 => "Data_block_2".y1, out2 => "Data_block_2".y2)
   END_RUNG
   // the same network as SCL:
   "DI_blokFunkcyjny_A10"(in1 := "zmienna1",   // "blokFunkcyjny"
                          in2 := "Data_block_1".a1,
                          superZmienna := "superZmienna",
                          out1 => "Data_block_2".y1,
                          out2 => "Data_block_2".y2);
END_REGION

REGION Network 62: bardzo ważny komentarz
   RUNG wire#powerrail
      "DI_blokFunkcyjny_A10"(in1 := "zmienna1", in2 := "Data_block_1".a1, superZmienna := "superZmienna", out1 => "Data_block_2".y1, out2 => "Data_block_2".y2)
   END_RUNG
   // the same network as SCL:
   "DI_blokFunkcyjny_A10"(in1 := "zmienna1",   // "blokFunkcyjny"
                          in2 := "Data_block_1".a1,
                          superZmienna := "superZmienna",
                          out1 => "Data_block_2".y1,
                          out2 => "Data_block_2".y2);
END_REGION

REGION Network 63: bardzo ważny komentarz
   RUNG wire#powerrail
      "DI_blokFunkcyjny_A10"(in1 := "zmienna1", in2 := "Data_block_1".a1, superZmienna := "superZmienna", out1 => "Data_block_2".y1, out2 => "Data_block_2".y2)
   END_RUNG
   // the same network as SCL:
   "DI_blokFunkcyjny_A10"(in1 := "zmienna1",   // "blokFunkcyjny"
                          in2 := "Data_block_1".a1,
                          superZmienna := "superZmienna",
                          out1 => "Data_block_2".y1,
                          out2 => "Data_block_2".y2);
END_REGION

REGION Network 64: bardzo ważny komentarz
   RUNG wire#powerrail
      "DI_blokFunkcyjny_A10"(in1 := "zmienna1", in2 := "Data_block_1".a1, superZmienna := "superZmienna", out1 => "Data_block_2".y1, out2 => "Data_block_2".y2)
   END_RUNG
   // the same network as SCL:
   "DI_blokFunkcyjny_A10"(in1 := "zmienna1",   // "blokFunkcyjny"
                          in2 := "Data_block_1".a1,
                          superZmienna := "superZmienna",
                          out1 => "Data_block_2".y1,
                          out2 => "Data_block_2".y2);
END_REGION

REGION Network 65: bardzo ważny komentarz
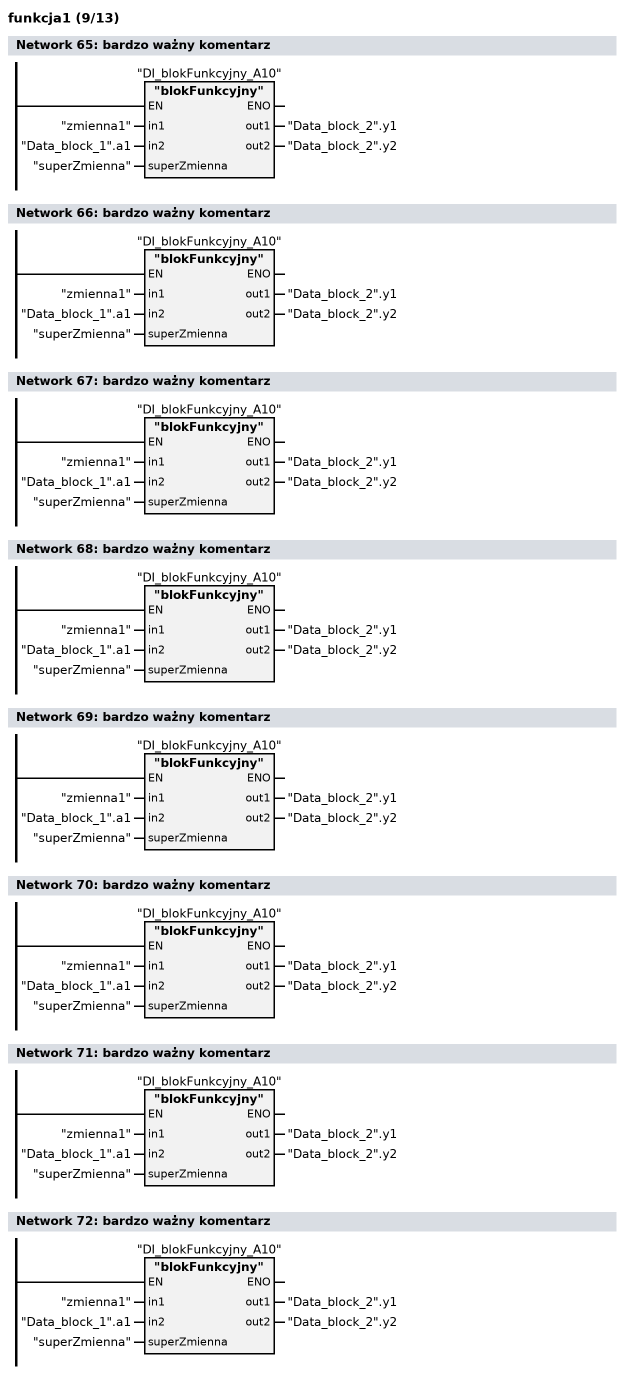
   RUNG wire#powerrail
      "DI_blokFunkcyjny_A10"(in1 := "zmienna1", in2 := "Data_block_1".a1, superZmienna := "superZmienna", out1 => "Data_block_2".y1, out2 => "Data_block_2".y2)
   END_RUNG
   // the same network as SCL:
   "DI_blokFunkcyjny_A10"(in1 := "zmienna1",   // "blokFunkcyjny"
                          in2 := "Data_block_1".a1,
                          superZmienna := "superZmienna",
                          out1 => "Data_block_2".y1,
                          out2 => "Data_block_2".y2);
END_REGION

REGION Network 66: bardzo ważny komentarz
   RUNG wire#powerrail
      "DI_blokFunkcyjny_A10"(in1 := "zmienna1", in2 := "Data_block_1".a1, superZmienna := "superZmienna", out1 => "Data_block_2".y1, out2 => "Data_block_2".y2)
   END_RUNG
   // the same network as SCL:
   "DI_blokFunkcyjny_A10"(in1 := "zmienna1",   // "blokFunkcyjny"
                          in2 := "Data_block_1".a1,
                          superZmienna := "superZmienna",
                          out1 => "Data_block_2".y1,
                          out2 => "Data_block_2".y2);
END_REGION

REGION Network 67: bardzo ważny komentarz
   RUNG wire#powerrail
      "DI_blokFunkcyjny_A10"(in1 := "zmienna1", in2 := "Data_block_1".a1, superZmienna := "superZmienna", out1 => "Data_block_2".y1, out2 => "Data_block_2".y2)
   END_RUNG
   // the same network as SCL:
   "DI_blokFunkcyjny_A10"(in1 := "zmienna1",   // "blokFunkcyjny"
                          in2 := "Data_block_1".a1,
                          superZmienna := "superZmienna",
                          out1 => "Data_block_2".y1,
                          out2 => "Data_block_2".y2);
END_REGION

REGION Network 68: bardzo ważny komentarz
   RUNG wire#powerrail
      "DI_blokFunkcyjny_A10"(in1 := "zmienna1", in2 := "Data_block_1".a1, superZmienna := "superZmienna", out1 => "Data_block_2".y1, out2 => "Data_block_2".y2)
   END_RUNG
   // the same network as SCL:
   "DI_blokFunkcyjny_A10"(in1 := "zmienna1",   // "blokFunkcyjny"
                          in2 := "Data_block_1".a1,
                          superZmienna := "superZmienna",
                          out1 => "Data_block_2".y1,
                          out2 => "Data_block_2".y2);
END_REGION

REGION Network 69: bardzo ważny komentarz
   RUNG wire#powerrail
      "DI_blokFunkcyjny_A10"(in1 := "zmienna1", in2 := "Data_block_1".a1, superZmienna := "superZmienna", out1 => "Data_block_2".y1, out2 => "Data_block_2".y2)
   END_RUNG
   // the same network as SCL:
   "DI_blokFunkcyjny_A10"(in1 := "zmienna1",   // "blokFunkcyjny"
                          in2 := "Data_block_1".a1,
                          superZmienna := "superZmienna",
                          out1 => "Data_block_2".y1,
                          out2 => "Data_block_2".y2);
END_REGION

REGION Network 70: bardzo ważny komentarz
   RUNG wire#powerrail
      "DI_blokFunkcyjny_A10"(in1 := "zmienna1", in2 := "Data_block_1".a1, superZmienna := "superZmienna", out1 => "Data_block_2".y1, out2 => "Data_block_2".y2)
   END_RUNG
   // the same network as SCL:
   "DI_blokFunkcyjny_A10"(in1 := "zmienna1",   // "blokFunkcyjny"
                          in2 := "Data_block_1".a1,
                          superZmienna := "superZmienna",
                          out1 => "Data_block_2".y1,
                          out2 => "Data_block_2".y2);
END_REGION

REGION Network 71: bardzo ważny komentarz
   RUNG wire#powerrail
      "DI_blokFunkcyjny_A10"(in1 := "zmienna1", in2 := "Data_block_1".a1, superZmienna := "superZmienna", out1 => "Data_block_2".y1, out2 => "Data_block_2".y2)
   END_RUNG
   // the same network as SCL:
   "DI_blokFunkcyjny_A10"(in1 := "zmienna1",   // "blokFunkcyjny"
                          in2 := "Data_block_1".a1,
                          superZmienna := "superZmienna",
                          out1 => "Data_block_2".y1,
                          out2 => "Data_block_2".y2);
END_REGION

REGION Network 72: bardzo ważny komentarz
   RUNG wire#powerrail
      "DI_blokFunkcyjny_A10"(in1 := "zmienna1", in2 := "Data_block_1".a1, superZmienna := "superZmienna", out1 => "Data_block_2".y1, out2 => "Data_block_2".y2)
   END_RUNG
   // the same network as SCL:
   "DI_blokFunkcyjny_A10"(in1 := "zmienna1",   // "blokFunkcyjny"
                          in2 := "Data_block_1".a1,
                          superZmienna := "superZmienna",
                          out1 => "Data_block_2".y1,
                          out2 => "Data_block_2".y2);
END_REGION

REGION Network 73: bardzo ważny komentarz
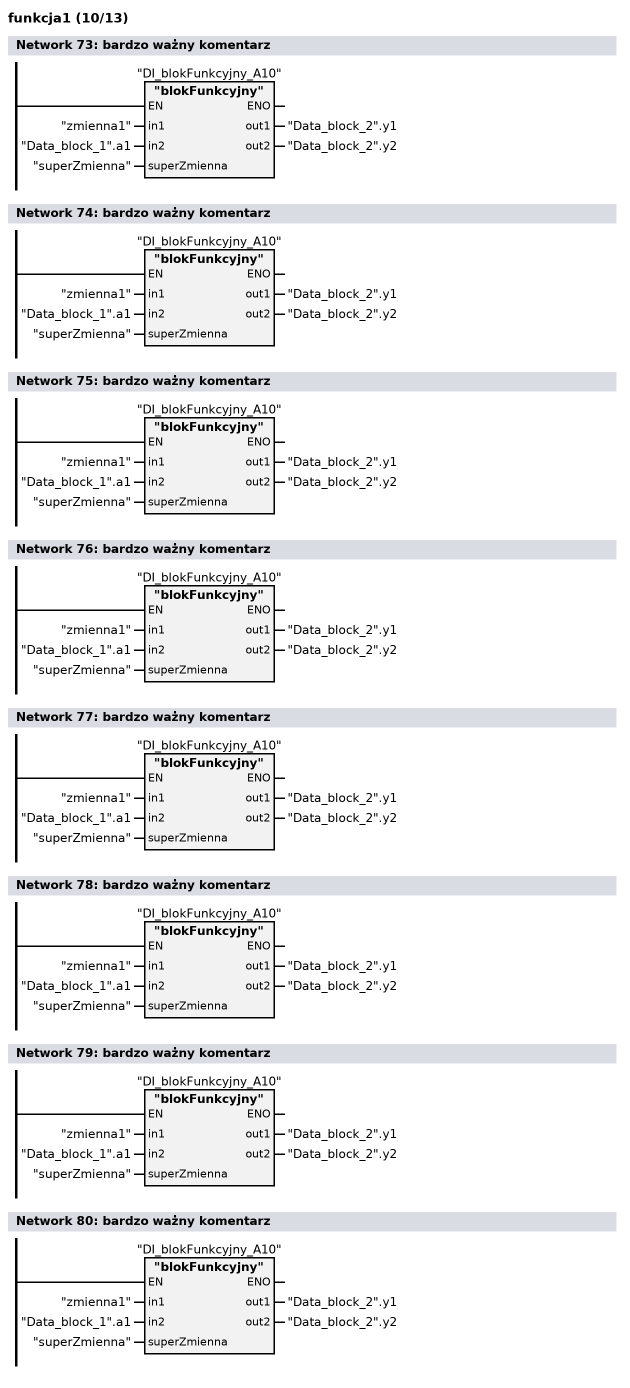
   RUNG wire#powerrail
      "DI_blokFunkcyjny_A10"(in1 := "zmienna1", in2 := "Data_block_1".a1, superZmienna := "superZmienna", out1 => "Data_block_2".y1, out2 => "Data_block_2".y2)
   END_RUNG
   // the same network as SCL:
   "DI_blokFunkcyjny_A10"(in1 := "zmienna1",   // "blokFunkcyjny"
                          in2 := "Data_block_1".a1,
                          superZmienna := "superZmienna",
                          out1 => "Data_block_2".y1,
                          out2 => "Data_block_2".y2);
END_REGION

REGION Network 74: bardzo ważny komentarz
   RUNG wire#powerrail
      "DI_blokFunkcyjny_A10"(in1 := "zmienna1", in2 := "Data_block_1".a1, superZmienna := "superZmienna", out1 => "Data_block_2".y1, out2 => "Data_block_2".y2)
   END_RUNG
   // the same network as SCL:
   "DI_blokFunkcyjny_A10"(in1 := "zmienna1",   // "blokFunkcyjny"
                          in2 := "Data_block_1".a1,
                          superZmienna := "superZmienna",
                          out1 => "Data_block_2".y1,
                          out2 => "Data_block_2".y2);
END_REGION

REGION Network 75: bardzo ważny komentarz
   RUNG wire#powerrail
      "DI_blokFunkcyjny_A10"(in1 := "zmienna1", in2 := "Data_block_1".a1, superZmienna := "superZmienna", out1 => "Data_block_2".y1, out2 => "Data_block_2".y2)
   END_RUNG
   // the same network as SCL:
   "DI_blokFunkcyjny_A10"(in1 := "zmienna1",   // "blokFunkcyjny"
                          in2 := "Data_block_1".a1,
                          superZmienna := "superZmienna",
                          out1 => "Data_block_2".y1,
                          out2 => "Data_block_2".y2);
END_REGION

REGION Network 76: bardzo ważny komentarz
   RUNG wire#powerrail
      "DI_blokFunkcyjny_A10"(in1 := "zmienna1", in2 := "Data_block_1".a1, superZmienna := "superZmienna", out1 => "Data_block_2".y1, out2 => "Data_block_2".y2)
   END_RUNG
   // the same network as SCL:
   "DI_blokFunkcyjny_A10"(in1 := "zmienna1",   // "blokFunkcyjny"
                          in2 := "Data_block_1".a1,
                          superZmienna := "superZmienna",
                          out1 => "Data_block_2".y1,
                          out2 => "Data_block_2".y2);
END_REGION

REGION Network 77: bardzo ważny komentarz
   RUNG wire#powerrail
      "DI_blokFunkcyjny_A10"(in1 := "zmienna1", in2 := "Data_block_1".a1, superZmienna := "superZmienna", out1 => "Data_block_2".y1, out2 => "Data_block_2".y2)
   END_RUNG
   // the same network as SCL:
   "DI_blokFunkcyjny_A10"(in1 := "zmienna1",   // "blokFunkcyjny"
                          in2 := "Data_block_1".a1,
                          superZmienna := "superZmienna",
                          out1 => "Data_block_2".y1,
                          out2 => "Data_block_2".y2);
END_REGION

REGION Network 78: bardzo ważny komentarz
   RUNG wire#powerrail
      "DI_blokFunkcyjny_A10"(in1 := "zmienna1", in2 := "Data_block_1".a1, superZmienna := "superZmienna", out1 => "Data_block_2".y1, out2 => "Data_block_2".y2)
   END_RUNG
   // the same network as SCL:
   "DI_blokFunkcyjny_A10"(in1 := "zmienna1",   // "blokFunkcyjny"
                          in2 := "Data_block_1".a1,
                          superZmienna := "superZmienna",
                          out1 => "Data_block_2".y1,
                          out2 => "Data_block_2".y2);
END_REGION

REGION Network 79: bardzo ważny komentarz
   RUNG wire#powerrail
      "DI_blokFunkcyjny_A10"(in1 := "zmienna1", in2 := "Data_block_1".a1, superZmienna := "superZmienna", out1 => "Data_block_2".y1, out2 => "Data_block_2".y2)
   END_RUNG
   // the same network as SCL:
   "DI_blokFunkcyjny_A10"(in1 := "zmienna1",   // "blokFunkcyjny"
                          in2 := "Data_block_1".a1,
                          superZmienna := "superZmienna",
                          out1 => "Data_block_2".y1,
                          out2 => "Data_block_2".y2);
END_REGION

REGION Network 80: bardzo ważny komentarz
   RUNG wire#powerrail
      "DI_blokFunkcyjny_A10"(in1 := "zmienna1", in2 := "Data_block_1".a1, superZmienna := "superZmienna", out1 => "Data_block_2".y1, out2 => "Data_block_2".y2)
   END_RUNG
   // the same network as SCL:
   "DI_blokFunkcyjny_A10"(in1 := "zmienna1",   // "blokFunkcyjny"
                          in2 := "Data_block_1".a1,
                          superZmienna := "superZmienna",
                          out1 => "Data_block_2".y1,
                          out2 => "Data_block_2".y2);
END_REGION

REGION Network 81: bardzo ważny komentarz
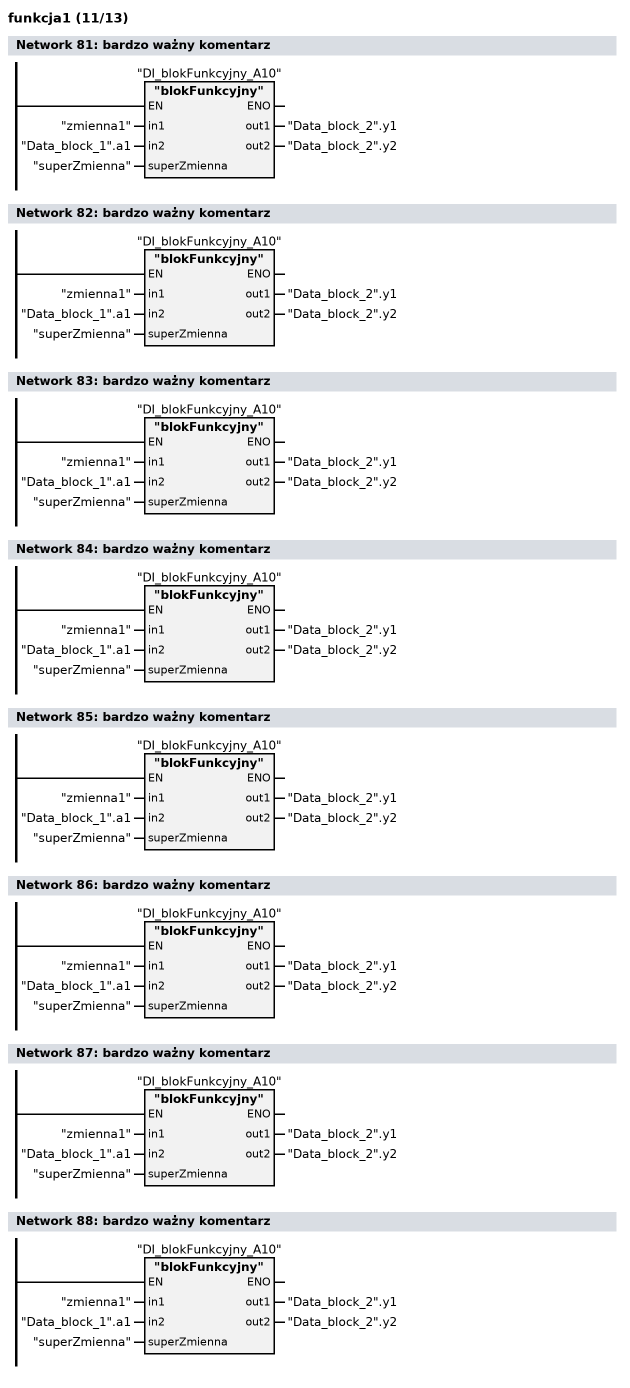
   RUNG wire#powerrail
      "DI_blokFunkcyjny_A10"(in1 := "zmienna1", in2 := "Data_block_1".a1, superZmienna := "superZmienna", out1 => "Data_block_2".y1, out2 => "Data_block_2".y2)
   END_RUNG
   // the same network as SCL:
   "DI_blokFunkcyjny_A10"(in1 := "zmienna1",   // "blokFunkcyjny"
                          in2 := "Data_block_1".a1,
                          superZmienna := "superZmienna",
                          out1 => "Data_block_2".y1,
                          out2 => "Data_block_2".y2);
END_REGION

REGION Network 82: bardzo ważny komentarz
   RUNG wire#powerrail
      "DI_blokFunkcyjny_A10"(in1 := "zmienna1", in2 := "Data_block_1".a1, superZmienna := "superZmienna", out1 => "Data_block_2".y1, out2 => "Data_block_2".y2)
   END_RUNG
   // the same network as SCL:
   "DI_blokFunkcyjny_A10"(in1 := "zmienna1",   // "blokFunkcyjny"
                          in2 := "Data_block_1".a1,
                          superZmienna := "superZmienna",
                          out1 => "Data_block_2".y1,
                          out2 => "Data_block_2".y2);
END_REGION

REGION Network 83: bardzo ważny komentarz
   RUNG wire#powerrail
      "DI_blokFunkcyjny_A10"(in1 := "zmienna1", in2 := "Data_block_1".a1, superZmienna := "superZmienna", out1 => "Data_block_2".y1, out2 => "Data_block_2".y2)
   END_RUNG
   // the same network as SCL:
   "DI_blokFunkcyjny_A10"(in1 := "zmienna1",   // "blokFunkcyjny"
                          in2 := "Data_block_1".a1,
                          superZmienna := "superZmienna",
                          out1 => "Data_block_2".y1,
                          out2 => "Data_block_2".y2);
END_REGION

REGION Network 84: bardzo ważny komentarz
   RUNG wire#powerrail
      "DI_blokFunkcyjny_A10"(in1 := "zmienna1", in2 := "Data_block_1".a1, superZmienna := "superZmienna", out1 => "Data_block_2".y1, out2 => "Data_block_2".y2)
   END_RUNG
   // the same network as SCL:
   "DI_blokFunkcyjny_A10"(in1 := "zmienna1",   // "blokFunkcyjny"
                          in2 := "Data_block_1".a1,
                          superZmienna := "superZmienna",
                          out1 => "Data_block_2".y1,
                          out2 => "Data_block_2".y2);
END_REGION

REGION Network 85: bardzo ważny komentarz
   RUNG wire#powerrail
      "DI_blokFunkcyjny_A10"(in1 := "zmienna1", in2 := "Data_block_1".a1, superZmienna := "superZmienna", out1 => "Data_block_2".y1, out2 => "Data_block_2".y2)
   END_RUNG
   // the same network as SCL:
   "DI_blokFunkcyjny_A10"(in1 := "zmienna1",   // "blokFunkcyjny"
                          in2 := "Data_block_1".a1,
                          superZmienna := "superZmienna",
                          out1 => "Data_block_2".y1,
                          out2 => "Data_block_2".y2);
END_REGION

REGION Network 86: bardzo ważny komentarz
   RUNG wire#powerrail
      "DI_blokFunkcyjny_A10"(in1 := "zmienna1", in2 := "Data_block_1".a1, superZmienna := "superZmienna", out1 => "Data_block_2".y1, out2 => "Data_block_2".y2)
   END_RUNG
   // the same network as SCL:
   "DI_blokFunkcyjny_A10"(in1 := "zmienna1",   // "blokFunkcyjny"
                          in2 := "Data_block_1".a1,
                          superZmienna := "superZmienna",
                          out1 => "Data_block_2".y1,
                          out2 => "Data_block_2".y2);
END_REGION

REGION Network 87: bardzo ważny komentarz
   RUNG wire#powerrail
      "DI_blokFunkcyjny_A10"(in1 := "zmienna1", in2 := "Data_block_1".a1, superZmienna := "superZmienna", out1 => "Data_block_2".y1, out2 => "Data_block_2".y2)
   END_RUNG
   // the same network as SCL:
   "DI_blokFunkcyjny_A10"(in1 := "zmienna1",   // "blokFunkcyjny"
                          in2 := "Data_block_1".a1,
                          superZmienna := "superZmienna",
                          out1 => "Data_block_2".y1,
                          out2 => "Data_block_2".y2);
END_REGION

REGION Network 88: bardzo ważny komentarz
   RUNG wire#powerrail
      "DI_blokFunkcyjny_A10"(in1 := "zmienna1", in2 := "Data_block_1".a1, superZmienna := "superZmienna", out1 => "Data_block_2".y1, out2 => "Data_block_2".y2)
   END_RUNG
   // the same network as SCL:
   "DI_blokFunkcyjny_A10"(in1 := "zmienna1",   // "blokFunkcyjny"
                          in2 := "Data_block_1".a1,
                          superZmienna := "superZmienna",
                          out1 => "Data_block_2".y1,
                          out2 => "Data_block_2".y2);
END_REGION

REGION Network 89: bardzo ważny komentarz
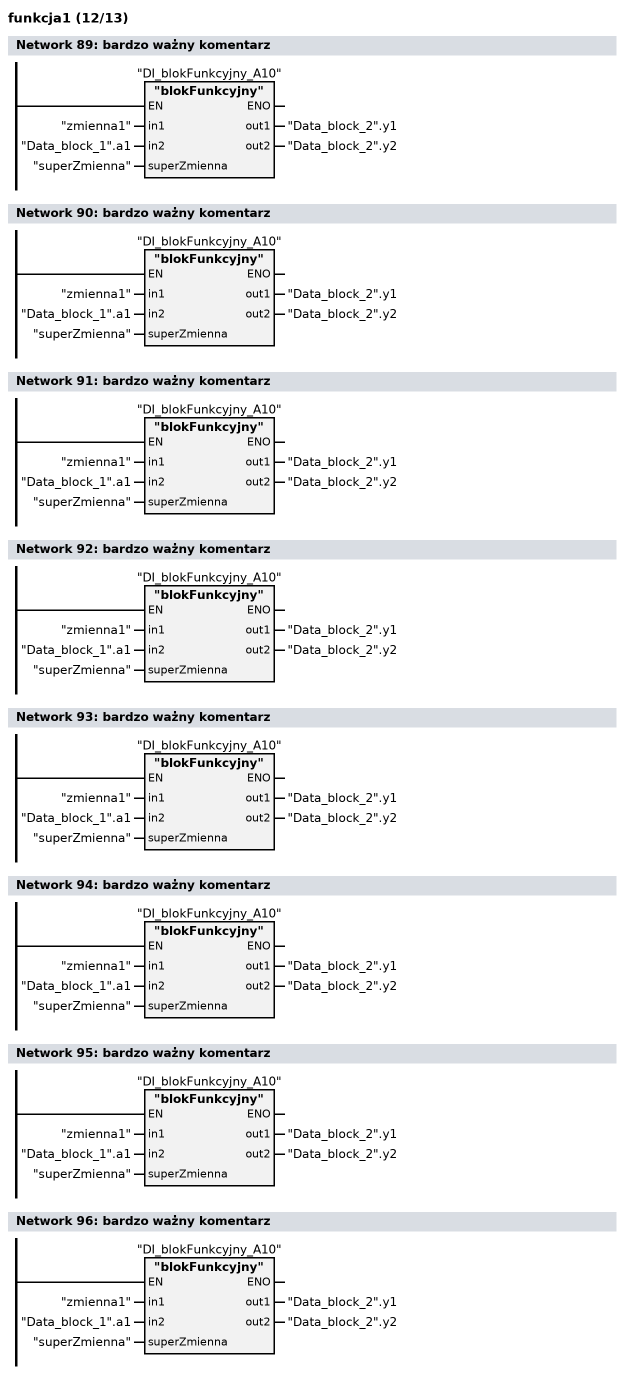
   RUNG wire#powerrail
      "DI_blokFunkcyjny_A10"(in1 := "zmienna1", in2 := "Data_block_1".a1, superZmienna := "superZmienna", out1 => "Data_block_2".y1, out2 => "Data_block_2".y2)
   END_RUNG
   // the same network as SCL:
   "DI_blokFunkcyjny_A10"(in1 := "zmienna1",   // "blokFunkcyjny"
                          in2 := "Data_block_1".a1,
                          superZmienna := "superZmienna",
                          out1 => "Data_block_2".y1,
                          out2 => "Data_block_2".y2);
END_REGION

REGION Network 90: bardzo ważny komentarz
   RUNG wire#powerrail
      "DI_blokFunkcyjny_A10"(in1 := "zmienna1", in2 := "Data_block_1".a1, superZmienna := "superZmienna", out1 => "Data_block_2".y1, out2 => "Data_block_2".y2)
   END_RUNG
   // the same network as SCL:
   "DI_blokFunkcyjny_A10"(in1 := "zmienna1",   // "blokFunkcyjny"
                          in2 := "Data_block_1".a1,
                          superZmienna := "superZmienna",
                          out1 => "Data_block_2".y1,
                          out2 => "Data_block_2".y2);
END_REGION

REGION Network 91: bardzo ważny komentarz
   RUNG wire#powerrail
      "DI_blokFunkcyjny_A10"(in1 := "zmienna1", in2 := "Data_block_1".a1, superZmienna := "superZmienna", out1 => "Data_block_2".y1, out2 => "Data_block_2".y2)
   END_RUNG
   // the same network as SCL:
   "DI_blokFunkcyjny_A10"(in1 := "zmienna1",   // "blokFunkcyjny"
                          in2 := "Data_block_1".a1,
                          superZmienna := "superZmienna",
                          out1 => "Data_block_2".y1,
                          out2 => "Data_block_2".y2);
END_REGION

REGION Network 92: bardzo ważny komentarz
   RUNG wire#powerrail
      "DI_blokFunkcyjny_A10"(in1 := "zmienna1", in2 := "Data_block_1".a1, superZmienna := "superZmienna", out1 => "Data_block_2".y1, out2 => "Data_block_2".y2)
   END_RUNG
   // the same network as SCL:
   "DI_blokFunkcyjny_A10"(in1 := "zmienna1",   // "blokFunkcyjny"
                          in2 := "Data_block_1".a1,
                          superZmienna := "superZmienna",
                          out1 => "Data_block_2".y1,
                          out2 => "Data_block_2".y2);
END_REGION

REGION Network 93: bardzo ważny komentarz
   RUNG wire#powerrail
      "DI_blokFunkcyjny_A10"(in1 := "zmienna1", in2 := "Data_block_1".a1, superZmienna := "superZmienna", out1 => "Data_block_2".y1, out2 => "Data_block_2".y2)
   END_RUNG
   // the same network as SCL:
   "DI_blokFunkcyjny_A10"(in1 := "zmienna1",   // "blokFunkcyjny"
                          in2 := "Data_block_1".a1,
                          superZmienna := "superZmienna",
                          out1 => "Data_block_2".y1,
                          out2 => "Data_block_2".y2);
END_REGION

REGION Network 94: bardzo ważny komentarz
   RUNG wire#powerrail
      "DI_blokFunkcyjny_A10"(in1 := "zmienna1", in2 := "Data_block_1".a1, superZmienna := "superZmienna", out1 => "Data_block_2".y1, out2 => "Data_block_2".y2)
   END_RUNG
   // the same network as SCL:
   "DI_blokFunkcyjny_A10"(in1 := "zmienna1",   // "blokFunkcyjny"
                          in2 := "Data_block_1".a1,
                          superZmienna := "superZmienna",
                          out1 => "Data_block_2".y1,
                          out2 => "Data_block_2".y2);
END_REGION

REGION Network 95: bardzo ważny komentarz
   RUNG wire#powerrail
      "DI_blokFunkcyjny_A10"(in1 := "zmienna1", in2 := "Data_block_1".a1, superZmienna := "superZmienna", out1 => "Data_block_2".y1, out2 => "Data_block_2".y2)
   END_RUNG
   // the same network as SCL:
   "DI_blokFunkcyjny_A10"(in1 := "zmienna1",   // "blokFunkcyjny"
                          in2 := "Data_block_1".a1,
                          superZmienna := "superZmienna",
                          out1 => "Data_block_2".y1,
                          out2 => "Data_block_2".y2);
END_REGION

REGION Network 96: bardzo ważny komentarz
   RUNG wire#powerrail
      "DI_blokFunkcyjny_A10"(in1 := "zmienna1", in2 := "Data_block_1".a1, superZmienna := "superZmienna", out1 => "Data_block_2".y1, out2 => "Data_block_2".y2)
   END_RUNG
   // the same network as SCL:
   "DI_blokFunkcyjny_A10"(in1 := "zmienna1",   // "blokFunkcyjny"
                          in2 := "Data_block_1".a1,
                          superZmienna := "superZmienna",
                          out1 => "Data_block_2".y1,
                          out2 => "Data_block_2".y2);
END_REGION

REGION Network 97: bardzo ważny komentarz
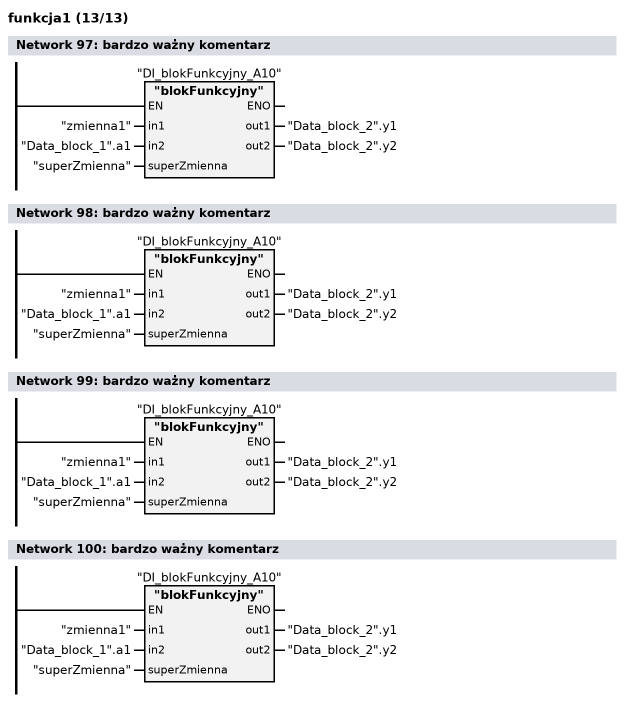
   RUNG wire#powerrail
      "DI_blokFunkcyjny_A10"(in1 := "zmienna1", in2 := "Data_block_1".a1, superZmienna := "superZmienna", out1 => "Data_block_2".y1, out2 => "Data_block_2".y2)
   END_RUNG
   // the same network as SCL:
   "DI_blokFunkcyjny_A10"(in1 := "zmienna1",   // "blokFunkcyjny"
                          in2 := "Data_block_1".a1,
                          superZmienna := "superZmienna",
                          out1 => "Data_block_2".y1,
                          out2 => "Data_block_2".y2);
END_REGION

REGION Network 98: bardzo ważny komentarz
   RUNG wire#powerrail
      "DI_blokFunkcyjny_A10"(in1 := "zmienna1", in2 := "Data_block_1".a1, superZmienna := "superZmienna", out1 => "Data_block_2".y1, out2 => "Data_block_2".y2)
   END_RUNG
   // the same network as SCL:
   "DI_blokFunkcyjny_A10"(in1 := "zmienna1",   // "blokFunkcyjny"
                          in2 := "Data_block_1".a1,
                          superZmienna := "superZmienna",
                          out1 => "Data_block_2".y1,
                          out2 => "Data_block_2".y2);
END_REGION

REGION Network 99: bardzo ważny komentarz
   RUNG wire#powerrail
      "DI_blokFunkcyjny_A10"(in1 := "zmienna1", in2 := "Data_block_1".a1, superZmienna := "superZmienna", out1 => "Data_block_2".y1, out2 => "Data_block_2".y2)
   END_RUNG
   // the same network as SCL:
   "DI_blokFunkcyjny_A10"(in1 := "zmienna1",   // "blokFunkcyjny"
                          in2 := "Data_block_1".a1,
                          superZmienna := "superZmienna",
                          out1 => "Data_block_2".y1,
                          out2 => "Data_block_2".y2);
END_REGION

REGION Network 100: bardzo ważny komentarz
   RUNG wire#powerrail
      "DI_blokFunkcyjny_A10"(in1 := "zmienna1", in2 := "Data_block_1".a1, superZmienna := "superZmienna", out1 => "Data_block_2".y1, out2 => "Data_block_2".y2)
   END_RUNG
   // the same network as SCL:
   "DI_blokFunkcyjny_A10"(in1 := "zmienna1",   // "blokFunkcyjny"
                          in2 := "Data_block_1".a1,
                          superZmienna := "superZmienna",
                          out1 => "Data_block_2".y1,
                          out2 => "Data_block_2".y2);
END_REGION
END_FUNCTION
